{attribute 'qualified_only'}
{attribute 'strict'}
TYPE E_TagStatus :
(
	NotPresent	:= 0,
	FixCode		:= 1,
	UserCode	:= 2
)BYTE := NotPresent;
END_TYPE

(* stored: Version 1.1.0.1, ProductVersion 3.1.4024.11
   EnumerationTextList E_TagStatus: Id {59ca2db3-18b8-4c5d-af75-6ed4208e6e6d} *)
